FUNCTION_BLOCK T_RoboConnect_SetDigitalOutput_CorrectIndexPasses EXTENDS T_UnitTestBase
VAR
  robot : I_RoboConnect;
  targetDO : UINT;
  myTestState, prevState :
    (INIT, ARRANGE, ACT, ASSERT) := INIT;
  expected, actual : BOOL;
  counter : UINT;
END_VAR

CASE myTestState OF
  INIT:
    StateChanged();
    myTestState := ARRANGE;

  ARRANGE:
    IF StateChanged() THEN
      expected := TRUE;
      robot.Connect();
    END_IF

    IF robot.Connected THEN
      myTestState := ACT;
    END_IF

  ACT:
    actual := robot.SetDigitalOutput(targetDO, TRUE);
    myTestState := ASSERT;

  ASSERT:
    actual := robot.GetDigitalOutput(targetDO);
    assertion.AssertEquals_BOOL(expected, actual, 'actual := robot.SetDigitalOutput(targetDO, TRUE)');
    TestFinished();
    myTestState := INIT;

END_CASE

METHOD FB_init : BOOL
VAR_INPUT
  bInitRetains : BOOL; // if TRUE, the retain variables are initialized (warm start / cold start)
  bInCopyCode : BOOL; // if TRUE, the instance afterwards gets moved into the copy code (online change)
  TestSuite : tcl_SimpleUnitTestLibrary.I_TestSuite;
  robot : I_TcRobot;
  targetDo : UINT;
END_VAR
THIS^.robot := robot;
THIS^.targetDo := targetDo;
END_METHOD

METHOD PRIVATE StateChanged : BOOL
IF  myTestState = prevState THEN
  RETURN;
END_IF

prevState := myTestState;
StateChanged := TRUE;
END_METHOD

METHOD WaitForCycles : BOOL
VAR_INPUT
  maxCount : UINT;
END_VAR
counter := counter + 1;

IF counter = maxCount THEN
  counter := 0;
  WaitForCycles := TRUE;
END_IF
END_METHOD

END_FUNCTION_BLOCK

(* stored: Version 1.1.0.1
   POU T_TcRobot_SetDigitalOutput_CorrectIndexPasses: Id {b8d4cd31-bf48-43f0-8759-d7b73c8d87d5}, SpecialFunc None
   Method FB_init: Id {2d58c847-4f1a-4452-a0f2-cb97cd433616}
   Method StateChanged: Id {e2eeb13e-7e0d-4556-9f87-206f7e5662c4}
   Method WaitForCycles: Id {39e6bd2f-ea92-4f22-937b-b1da8fc779d7} *)
